FUNCTION_BLOCK FB_TemperatureSensor EXTENDS FB_Sensor
VAR_INPUT
END_VAR
VAR_OUTPUT
	fTemperature : REAL; //measured temperature in degreeC
END_VAR
VAR	
	//default parameters
	localDefaultParameters : ST_TemperatureSensorDefaultParameters;	

	//I/O-Links
	temperature_IN AT %I* : INT;
END_VAR

METHOD SetState_AI : BOOL
VAR_INPUT
END_VAR
VAR
END_VAR
// conversion with 0.01 resolution
fTemperature := (INT_TO_REAL(temperature_IN))*0.01;

//sensor state
sensorState.fValue := fTemperature;
sensorState.sUnit := localDefaultParameters.sUnit;
END_METHOD

PROPERTY ST_DefaultParameters : REFERENCE TO ST_TemperatureSensorDefaultParameters
SET
localDefaultParameters := ST_DefaultParameters;
END_SET
END_PROPERTY

END_FUNCTION_BLOCK

(* stored: Version 1.1.0.1, ProductVersion 3.1.4024.9
   POU FB_TemperatureSensor: Id {5862196d-9579-4df5-99e3-f378128664c6}, SpecialFunc None
   Method SetState_AI: Id {0a841d63-6fae-4c9e-a077-b7b01fa6149c}
   Property ST_DefaultParameters: Id {5d8d5df2-304d-42ad-ad33-aa6063b91df0}
   Set Set: Id {7de6bca6-54f7-41a1-b870-78a80dba2c53} *)
